// TIA Portal V16 export
// export: Created 2023-03-29T11:05:04.7441942Z, ExportSetting WithDefaults, DisplayName Totally Integrated Automation Portal, DisplayVersion V16 Update 6, DisplayName TIA Portal Version Control Interface, DisplayVersion V16 Update 2, DisplayName TIA Portal Openness, DisplayVersion V16 Update 6, DisplayName STEP 7 Professional, DisplayVersion V16 Update 6, DisplayName STEP 7 Safety, DisplayVersion V16, DisplayName WinCC Advanced, DisplayVersion V16 Update 6
VAR_GLOBAL   // PLC tag table "Sim"
   Sim_wiodaca AT %M1200.0 : Bool;
   Sim_SetUp_M25 AT %M1200.1 : Bool;
   Sim_SetDown_M25 AT %M1200.2 : Bool;
   Sim_aut_man AT %M1200.4 : Bool;
   Sim_SetDown_M27 AT %M1200.5 : Bool;
   simAnalogB5_Increm AT %M1041.0 : Bool;
   simAnalogB5_load AT %M1041.1 : Bool;
   simAnalogB5_Licznik AT %MW1042 : Word;
   simAnalogB5_decrem AT %M1041.4 : Bool;
   Tag_Start1 AT %M1041.2 : Bool;
   Tag_Start2 AT %M1041.3 : Bool;
   i AT %M1041.5 : Bool;
   Sim_daneMW AT %MD2000 : Real;
   "Ustaw alarm P3" AT %M1040.4 : Bool;
   STP_funkction_1 AT %M1041.7 : Bool;
   STP_funkction AT %M1041.6 : Bool;
   Sim_WarningHbar AT %M1200.3 : Bool;
END_VAR
